INTERFACE I_Comm

METHOD Publish : BOOL
VAR_INPUT
	domain			: STRING(255) := 'environment';
	location		: STRING(255) := 'roof';
	parameter		: STRING(255);
	value			: STRING(255);	
END_VAR
VAR_OUTPUT
	published	: BOOL;
END_VAR
END_METHOD

METHOD PublishLog : BOOL
VAR_INPUT
	level		: STRING(255) := 'INFO';
	message		: STRING(255);	
END_VAR
VAR_OUTPUT
	published	: BOOL;
END_VAR
END_METHOD

END_INTERFACE

(* stored: Version 1.1.0.1, ProductVersion 3.1.4024.15
   Itf I_Comm: Id {aef8fd82-119a-49b9-85f1-c62ccf3b36f3}
   Method Publish: Id {5b2a42b4-e26b-405d-99ca-66788602b2d5}
   Method PublishLog: Id {bb17fd3c-9433-4b30-9d10-3bf6aa5dc9fe} *)
